{attribute 'qualified_only'}
VAR_GLOBAL
	
	enableAxi: BOOL;
	runFWD: BOOL;
	resetAxi: BOOL;
	revs: REAL;
	mL_target: REAL;
	runBWD: BOOL;
	enableValv: BOOL;
	valvPos: INT;
END_VAR

(* stored: Version 1.1.0.1, ProductVersion 3.1.4024.12
   GVL GVL_Marco: Id {80397fe9-0a64-47cf-a8bc-5c0cd05c5f13} *)
